(* IEC 61131-3 sources: repolevel_ST_code_completion/output/full_case_fixed/repoeval_Proxy_Application/readful_result_history, 6 files *)

(* ---- Proxy_0.st ---- *)
{attribute 'enable_dynamic_creation'}
FUNCTION_BLOCK Proxy IMPLEMENTS  Subject_Interface
VAR_INPUT
END_VAR
VAR_OUTPUT
END_VAR
VAR
    refToRealSubject : POINTER TO Realsubject;
    iTempPassword : INT;
END_VAR
VAR_STAT
    iRealPassword : INT := 1234;
END_VAR

METHOD fb_init
VAR_INPUT
    bInitRetains : BOOL;
    bInCopyCode : BOOL;
    ptrToRealSubject : POINTER TO Realsubject;
END_VAR
VAR_OUTPUT
END_VAR
VAR
END_VAR
refToRealSubject := ptrToRealSubject;

METHOD Get_Method : INT
VAR_INPUT
END_VAR
IF iTempPassword = iRealPassword THEN
    RETURN refToRealSubject^.iProp;
ELSE
    RETURN -1; // Invalid password
END_IF;

METHOD Set_Method
VAR_INPUT
    num : INT;
END_VAR
IF iTempPassword = iRealPassword THEN
    refToRealSubject^.iProp := num;
END_IF;
END_FUNCTION_BLOCK

(* ---- Proxy_2.st ---- *)
{attribute 'enable_dynamic_creation'}
FUNCTION_BLOCK Proxy IMPLEMENTS  Subject_Interface
VAR_INPUT
END_VAR
VAR_OUTPUT
END_VAR
VAR
    refToRealSubject : POINTER TO Realsubject;
    iTempPassword : INT;
END_VAR
VAR_STAT
    iRealPassword : INT := 1234;
END_VAR

METHOD fb_init
VAR_INPUT
  bInitRetains : BOOL;
  bInCopyCode : BOOL;
  ptrToRealSubject : POINTER TO Realsubject;
END_VAR
VAR_OUTPUT
END_VAR
VAR
END_VAR
IF ptrToRealSubject <> 0 THEN
  refToRealSubject := ptrToRealSubject;
END_IF;

METHOD Get_Method : INT
VAR_INPUT
END_VAR
IF iTempPassword = iRealPassword THEN
  IF refToRealSubject <> 0 THEN
    RETURN refToRealSubject^.iProp;
  ELSE
    RETURN -1; // Invalid reference
  END_IF;
ELSE
  RETURN -1; // Invalid password
END_IF;

METHOD Set_Method
VAR_INPUT
  num : INT;
END_VAR
IF iTempPassword = iRealPassword THEN
  IF refToRealSubject <> 0 THEN
    refToRealSubject^.iProp := num;
  END_IF;
END_IF;
END_FUNCTION_BLOCK

(* ---- Realsubject_0.st ---- *)
{attribute 'enable_dynamic_creation'}
FUNCTION_BLOCK Realsubject IMPLEMENTS  Subject_Interface
VAR_INPUT
END_VAR
VAR_OUTPUT
END_VAR
VAR
    //Variable to get and set values
    iProp: INT;
END_VAR

METHOD Set_Method
VAR_INPUT
    num : INT; //Value to be set on the iProp variable
END_VAR
THIS^.iProp := num;

METHOD PUBLIC Get_Method : INT
VAR
END_VAR
Get_Method := THIS^.iProp;
END_FUNCTION_BLOCK

(* ---- Realsubject_1.st ---- *)
{attribute 'enable_dynamic_creation'}
FUNCTION_BLOCK Realsubject IMPLEMENTS  Subject_Interface
VAR_INPUT
END_VAR
VAR_OUTPUT
END_VAR
VAR
    //Variable to get and set values
    iProp: INT;
END_VAR

METHOD Set_Method
VAR_INPUT
  num : INT; //Value to be set on the iProp variable
END_VAR
iProp := num; // Assign directly, no need for a qualified reference

METHOD PUBLIC Get_Method : INT
VAR
END_VAR
RETURN iProp; // Return the value explicitly
END_FUNCTION_BLOCK

(* ---- Realsubject_2.st ---- *)
{attribute 'enable_dynamic_creation'}
FUNCTION_BLOCK Realsubject IMPLEMENTS  Subject_Interface
VAR_INPUT
END_VAR
VAR_OUTPUT
END_VAR
VAR
    //Variable to get and set values
    iProp: INT;
END_VAR

METHOD Set_Method
VAR_INPUT
 num : INT; //Value to be set on the iProp variable
END_VAR
iProp := num; // Assign directly, no need for a qualified reference
END_METHOD // Properly close the method

METHOD PUBLIC Get_Method : INT
VAR
END_VAR
RETURN iProp; // Return the value explicitly
END_METHOD // Properly close the method
END_FUNCTION_BLOCK

(* ---- Realsubject_3.st ---- *)
FUNCTION_BLOCK Realsubject IMPLEMENTS Subject_Interface
VAR_INPUT
END_VAR
VAR_OUTPUT
END_VAR
VAR
  //Variable to get and set values
  iProp: INT;
END_VAR

METHOD Set_Method
VAR_INPUT
num : INT; //Value to be set on the iProp variable
END_VAR
iProp := num; // Assign directly, no need for a qualified reference
END_METHOD // Properly close the method

METHOD PUBLIC Get_Method : INT
VAR
END_VAR
RETURN iProp; // Return the value explicitly
END_METHOD // Properly close the method
END_FUNCTION_BLOCK
